(* Logix 5000 project; controller ExampleWithCICD_L85E 1756-L85E rev 36.11; software revision 36.00 *)

TASK T00_MiscLogic (continuous, watchdog 500 ms) : P00_AND_OR_Logic, P01_ClearFault
TASK T01_ShowcaseDataTypes (periodic, rate 10 ms, priority 10, watchdog 500 ms) : P00_ShowcaseDataTypes

MODULES
   Local : 1756-L85E (ICP 0, rev 36.11)
END_MODULES

TYPE FAULTRECORD :
STRUCT
   Time_Low : DINT;   // Lower 32 bits of the fault timestamp value
   Time_High : DINT;   // Upper 32 bits of the fault timestamp value
   Type : INT;   // Fault type (program, I/O, and so forth)
   Code : INT;   // Unique code for the fault
   Info : DINT[8];   // Fault specific information
END_STRUCT
END_TYPE

VAR_GLOBAL   (* controller tags *)
   AT_ClearFault : BOOL;   // Automated Testing -------------------- clear the fault type & code
   AT_EnableIn : BOOL;   // Automated Testing -------------------- set the EnableIn AOI input parameter
   AT_FaultCode : DINT;   // Automated Testing -------------------- contains fault code number
   AT_FaultedIndicator : BOOL;   // Automated Testing -------------------- boolean HIGH if controller faulted
   AT_FaultType : DINT;   // Automated Testing -------------------- contains fault type number
   AT_ToggleTest : BOOL;   // Automated Testing -------------------- toggle to progress AOI testing by 1 clock cycle
   I_AND_1 : BOOL;   // AND Logic -------------------- input 1
   I_AND_2 : BOOL;   // AND Logic -------------------- input 2
   I_OR_1 : BOOL;   // OR Logic -------------------- input 1
   I_OR_2 : BOOL;   // OR Logic -------------------- input 2
   LowerBound_LINT : LINT := -9223372036854775808;
   LowerBound_REAL : REAL := -1.7976931e-38;
   LowerBound_STRING : STRING := 'Good Bye!';
   major_fault_record : FAULTRECORD;
   O_AND : BOOL;   // AND Logic -------------------- output
   O_OR : BOOL;   // OR Logic -------------------- output
   test2 : DINT;
   UpperBound_LINT : LINT := 9223372036854775807;
   UpperBound_REAL : REAL;
   UpperBound_STRING : STRING := 'Hello World!';
END_VAR

PROGRAM P00_AND_OR_Logic   (* main routine R00_Main *)

ROUTINE R00_Main   (* ladder *)
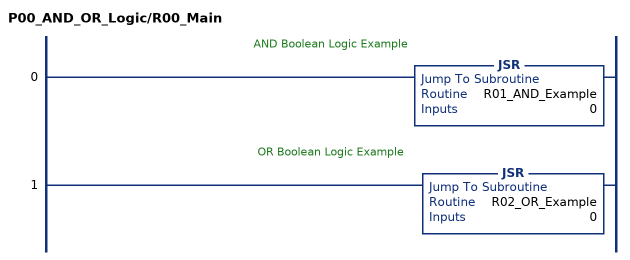
   // AND Boolean Logic Example
   0: JSR(R01_AND_Example,0);
   // OR Boolean Logic Example
   1: JSR(R02_OR_Example,0);
END_ROUTINE

ROUTINE R01_AND_Example   (* ladder *)
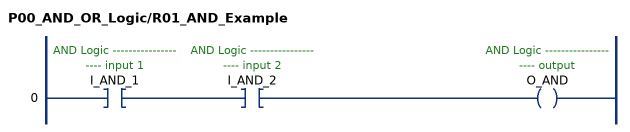
   0: XIC(I_AND_1)XIC(I_AND_2)OTE(O_AND);
END_ROUTINE

ROUTINE R02_OR_Example   (* ladder *)
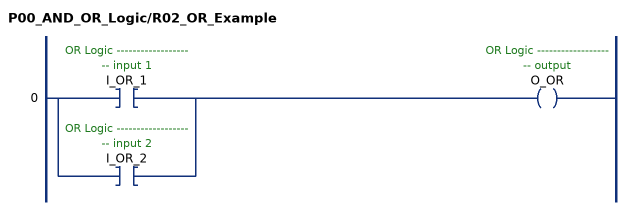
   0: [XIC(I_OR_1) ,XIC(I_OR_2) ]OTE(O_OR);
END_ROUTINE
END_PROGRAM

PROGRAM P00_ShowcaseDataTypes   (* main routine R00_ShowcaseDataTypes *)
VAR
   I_ToggleDINT_LocalTag : BOOL;
   I_ToggleEnable_LocalTag : BOOL;
   I_ToggleINT_LocalTag : BOOL;
   I_ToggleLINT_LocalTag : BOOL;
   I_ToggleREAL_LocalTag : BOOL;
   I_ToggleSINT_LocalTag : BOOL;
   I_ToggleSTRING_LocalTag : BOOL;
   O_DINT_LocalTag : DINT;
   O_INT_LocalTag : INT;
   O_LINT_LocalTag : LINT;
   O_REAL_LocalTag : REAL;
   O_SINT_LocalTag : SINT;
   O_STRING_LocalTag : STRING;
END_VAR

ROUTINE R00_ShowcaseDataTypes   (* ladder *)
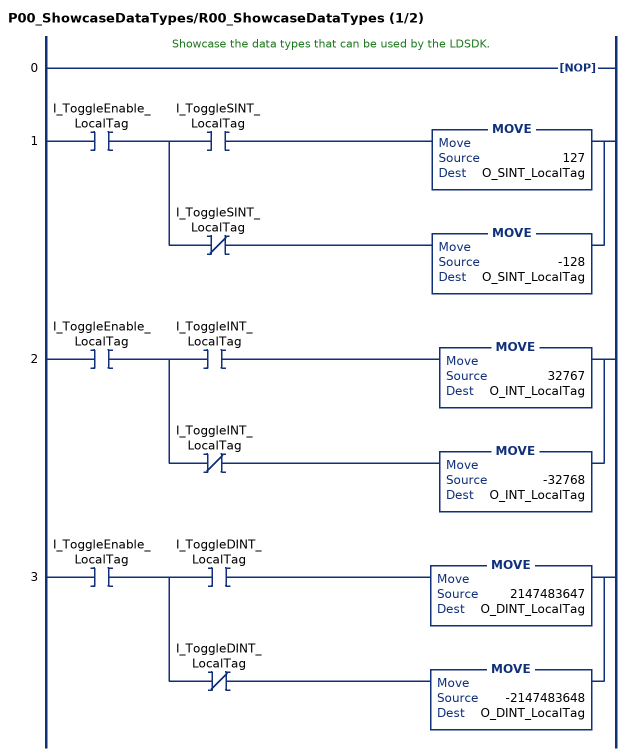
   // Showcase the data types that can be used by the LDSDK.
   0: NOP();
   1: XIC(I_ToggleEnable_LocalTag)[XIC(I_ToggleSINT_LocalTag) MOVE(127,O_SINT_LocalTag) ,XIO(I_ToggleSINT_LocalTag) MOVE(-128,O_SINT_LocalTag) ];
   2: XIC(I_ToggleEnable_LocalTag)[XIC(I_ToggleINT_LocalTag) MOVE(32767,O_INT_LocalTag) ,XIO(I_ToggleINT_LocalTag) MOVE(-32768,O_INT_LocalTag) ];
   3: XIC(I_ToggleEnable_LocalTag)[XIC(I_ToggleDINT_LocalTag) MOVE(2147483647,O_DINT_LocalTag) ,XIO(I_ToggleDINT_LocalTag) MOVE(-2147483648,O_DINT_LocalTag) ];
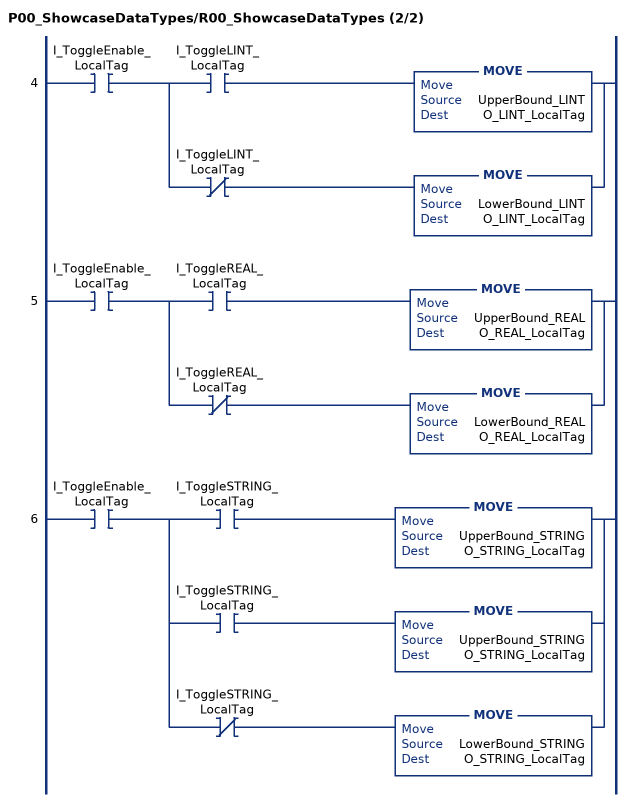
   4: XIC(I_ToggleEnable_LocalTag)[XIC(I_ToggleLINT_LocalTag) MOVE(UpperBound_LINT,O_LINT_LocalTag) ,XIO(I_ToggleLINT_LocalTag) MOVE(LowerBound_LINT,O_LINT_LocalTag) ];
   5: XIC(I_ToggleEnable_LocalTag)[XIC(I_ToggleREAL_LocalTag) MOVE(UpperBound_REAL,O_REAL_LocalTag) ,XIO(I_ToggleREAL_LocalTag) MOVE(LowerBound_REAL,O_REAL_LocalTag) ];
   6: XIC(I_ToggleEnable_LocalTag)[XIC(I_ToggleSTRING_LocalTag) MOVE(UpperBound_STRING,O_STRING_LocalTag) ,XIC(I_ToggleSTRING_LocalTag) MOVE(UpperBound_STRING,O_STRING_LocalTag) ,XIO(I_ToggleSTRING_LocalTag) MOVE(LowerBound_STRING,O_STRING_LocalTag) ];
END_ROUTINE
END_PROGRAM

PROGRAM P01_ClearFault   (* main routine R00_ClearFault *)

ROUTINE R00_ClearFault   (* ladder *)
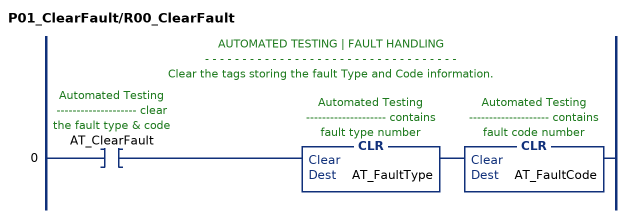
   // AUTOMATED TESTING | FAULT HANDLING
   // - - - - - - - - - - - - - - - - - - - - - - - - - - - - - - - - - -
   // Clear the tags storing the fault Type and Code information.
   0: XIC(AT_ClearFault)CLR(AT_FaultType)CLR(AT_FaultCode);
END_ROUTINE
END_PROGRAM

PROGRAM PXX_FaultHandler   (* main routine RXX_FaultHandler *)

ROUTINE RXX_FaultHandler   (* ladder *)
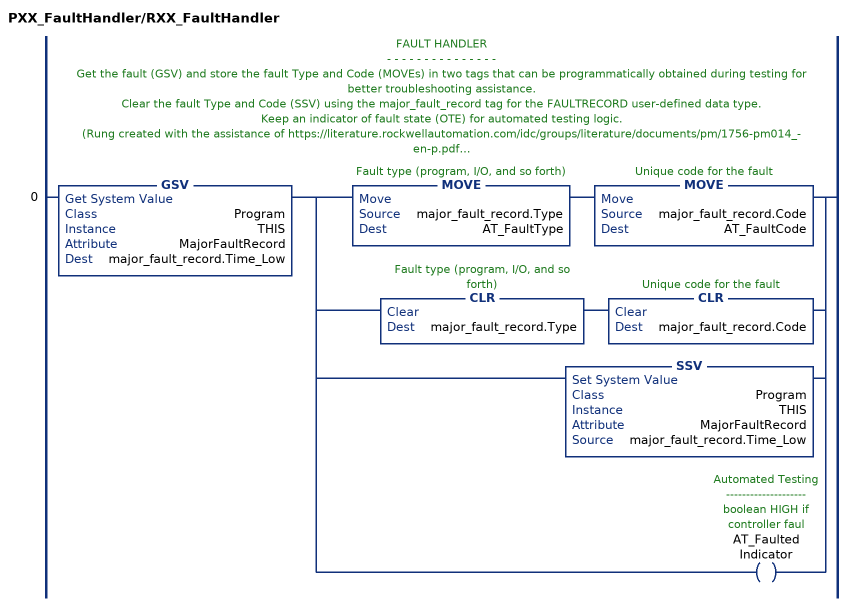
   // FAULT HANDLER
   // 													- - - - - - - - - - - - - - -
   // 													Get the fault (GSV) and store the fault Type and Code (MOVEs) in two tags that can be programmatically obtained during testing for better troubleshooting assistance.
   // 													Clear the fault Type and Code (SSV) using the major_fault_record tag for the FAULTRECORD user-defined data type.
   // 													Keep an indicator of fault state (OTE) for automated testing logic.
   // 													(Rung created with the assistance of https://literature.rockwellautomation.com/idc/groups/literature/documents/pm/1756-pm014_-en-p.pdf)
   // 													(Fault code spreadsheet link: https://literature.rockwellautomation.com/idc/groups/literature/documents/rd/1756-rd001_-en-p.xlsx)
   0: GSV(Program,THIS,MajorFaultRecord,major_fault_record.Time_Low)[MOVE(major_fault_record.Type,AT_FaultType) MOVE(major_fault_record.Code,AT_FaultCode) ,CLR(major_fault_record.Type) CLR(major_fault_record.Code) ,SSV(Program,THIS,MajorFaultRecord,major_fault_record.Time_Low) ,OTE(AT_FaultedIndicator) ];
END_ROUTINE
END_PROGRAM
